Universal Robots PolyScope program: Tall_LidToCamera.urp

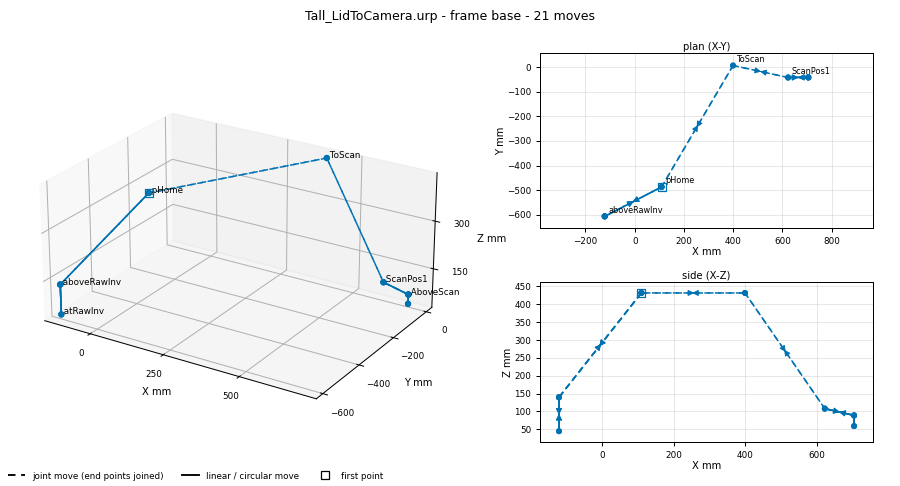
[picture p0: tool path of Tall_LidToCamera.urp in frame base, 21 of 21 moves have a stored position in this frame; points joined in program order, loops and branches not executed]
Program Tall_LidToCamera (installation=admin directory=/programs/THU_530PM/Final createdIn=3.8.0.61336 lastSavedIn=3.15.8.106339 robotSerialNumber=2015350926)
Calibrated DH parameters: a=[0, -0.425, -0.39225, 0, 0, 0]; d=[0.089159, 0, 0, 0.10915, 0.09465, 0.0823]; alpha=[1.570796, 0, 0, 1.570796, -1.570796, 0]; deltaTheta=[0, 0, 0, 0, 0, 0]
Robot Program (runOnlyOnce=true)
  Set DigitalOutput pin=digital_out[0]; digitalValue=0
  MoveJ speed 180 deg/s, acceleration 200 deg/s^2 (useActiveTCP=true)
    Waypoint pHome: TCP in base x=109.083 y=-486.882 z=431.849 mm, rx=0.0001 ry=3.1416 rz=-0.0001 rad; joints [89.992, -90.005, 90.008, -90.008, -90, -0.005] deg
    Call _adminLinearIndex3
    Waypoint aboveRawInv: TCP in base x=-121.783 y=-606.282 z=139.409 mm, rx=2.2212 ry=2.2177 rz=-0.0009 rad; joints [68.458, -61.32, 99.129, -127.902, -89.865, 68.547] deg
  MoveL speed 250 mm/s, acceleration 1200 mm/s^2 (useActiveTCP=true) feature=Base
    Waypoint atRawInv: TCP in base x=-121.765 y=-606.273 z=44.483 mm, rx=2.2211 ry=2.2178 rz=-0.0009 rad; joints [68.459, -52.315, 101.951, -139.731, -89.865, 68.544] deg
    Set DigitalOutput pin=digital_out[0]; digitalValue=1
    Wait Sleep waitTime=1
    Waypoint aboveRawInv: TCP in base x=-121.783 y=-606.282 z=139.409 mm, rx=2.2212 ry=2.2177 rz=-0.0009 rad; joints [68.458, -61.32, 99.129, -127.902, -89.865, 68.547] deg
  MoveJ speed 180 deg/s, acceleration 200 deg/s^2 (useActiveTCP=true)
    Waypoint pHome: TCP in base x=109.083 y=-486.882 z=431.849 mm, rx=0.0001 ry=3.1416 rz=-0.0001 rad; joints [89.992, -90.005, 90.008, -90.008, -90, -0.005] deg
  Call _adminLinearIndex1
  MoveJ speed 60 deg/s, acceleration 80 deg/s^2 (useActiveTCP=true)
    Waypoint ToScan: TCP in base x=399.431 y=6.288 z=431.784 mm, rx=0 ry=-3.1415 rz=0 rad; joints [165.046, -103.944, 102.123, -88.173, -90.001, 75.046] deg
    Waypoint ScanPos1: TCP in base x=623.056 y=-42.326 z=107.794 mm, rx=0.0456 ry=-3.1308 rz=0.0038 rad; joints [166.086, -57.904, 99.074, -130.624, -90.289, 74.42] deg
  MoveL speed 250 mm/s, acceleration 1200 mm/s^2 (useActiveTCP=true) feature=Base
    Waypoint AboveScan: TCP in base x=704.91 y=-41.789 z=88.68 mm, rx=0.0458 ry=-3.1307 rz=0.0039 rad; joints [167.748, -47.56, 83.623, -125.504, -90.275, 76.074] deg
    Waypoint AtScan: TCP in base x=704.921 y=-41.77 z=58.801 mm, rx=0.0456 ry=-3.1306 rz=0.0038 rad; joints [167.749, -45.085, 84.321, -128.675, -90.272, 76.08] deg
    Set DigitalOutput pin=digital_out[0]; digitalValue=0
    Wait Sleep waitTime=1
    Waypoint AboveScan: TCP in base x=704.91 y=-41.789 z=88.68 mm, rx=0.0458 ry=-3.1307 rz=0.0039 rad; joints [167.748, -47.56, 83.623, -125.504, -90.275, 76.074] deg
    Waypoint ScanPos1: TCP in base x=623.056 y=-42.326 z=107.794 mm, rx=0.0456 ry=-3.1308 rz=0.0038 rad; joints [166.086, -57.904, 99.074, -130.624, -90.289, 74.42] deg
    Script file /programs/THU_530PM/vision_pc_modbus.script
      | pc_ip = "10.241.34.37"
      | pc_port = 30002
      | 
      | connection = socket_open(pc_ip, pc_port, "vision_socket")
      | 
      | if (connection):
      |     socket_send_string("run_vision", "vision_socket")
      |     socket_close("vision_socket")
      | end
      | 
      | timeout = 15.0
      | elapsed =0.0
      | visionResult = 0
      | while visionResult == 0 and elapsed < timeout:
      |          sync()
      |          sleep(0.2)
      |          elapsed = elapsed + 0.2
      |          visionResult = modbus_get_signal_status ("vision_result")
      |          sync()
      | end
    Wait Sleep waitTime=2
  MoveJ speed 60 deg/s, acceleration 80 deg/s^2 (useActiveTCP=true)
    Waypoint AboveScan: TCP in base x=704.91 y=-41.789 z=88.68 mm, rx=0.0458 ry=-3.1307 rz=0.0039 rad; joints [167.748, -47.56, 83.623, -125.504, -90.275, 76.074] deg
    Waypoint AtScan: TCP in base x=704.921 y=-41.77 z=58.801 mm, rx=0.0456 ry=-3.1306 rz=0.0038 rad; joints [167.749, -45.085, 84.321, -128.675, -90.272, 76.08] deg
    Set DigitalOutput pin=digital_out[0]; digitalValue=1
    Wait Sleep waitTime=1
    Waypoint AboveScan: TCP in base x=704.91 y=-41.789 z=88.68 mm, rx=0.0458 ry=-3.1307 rz=0.0039 rad; joints [167.748, -47.56, 83.623, -125.504, -90.275, 76.074] deg
  MoveJ speed 60 deg/s, acceleration 80 deg/s^2 (useActiveTCP=true)
    Waypoint ScanPos1: TCP in base x=623.056 y=-42.326 z=107.794 mm, rx=0.0456 ry=-3.1308 rz=0.0038 rad; joints [166.086, -57.904, 99.074, -130.624, -90.289, 74.42] deg
    Waypoint ToScan: TCP in base x=399.431 y=6.288 z=431.784 mm, rx=0 ry=-3.1415 rz=0 rad; joints [165.046, -103.944, 102.123, -88.173, -90.001, 75.046] deg
    Waypoint pHome: TCP in base x=109.083 y=-486.882 z=431.849 mm, rx=0.0001 ry=3.1416 rz=-0.0001 rad; joints [89.992, -90.005, 90.008, -90.008, -90, -0.005] deg
    Call _adminLinearIndex3
    Waypoint aboveRawInv: TCP in base x=-121.783 y=-606.282 z=139.409 mm, rx=2.2212 ry=2.2177 rz=-0.0009 rad; joints [68.458, -61.32, 99.129, -127.902, -89.865, 68.547] deg
  MoveL speed 250 mm/s, acceleration 1200 mm/s^2 (useActiveTCP=true) feature=Base
    Waypoint atRawInv: TCP in base x=-121.765 y=-606.273 z=44.483 mm, rx=2.2211 ry=2.2178 rz=-0.0009 rad; joints [68.459, -52.315, 101.951, -139.731, -89.865, 68.544] deg
    Set DigitalOutput pin=digital_out[0]; digitalValue=0
    Wait Sleep waitTime=1
    Waypoint aboveRawInv: TCP in base x=-121.783 y=-606.282 z=139.409 mm, rx=2.2212 ry=2.2177 rz=-0.0009 rad; joints [68.458, -61.32, 99.129, -127.902, -89.865, 68.547] deg
  MoveJ speed 180 deg/s, acceleration 200 deg/s^2 (useActiveTCP=true)
    Waypoint pHome: TCP in base x=109.083 y=-486.882 z=431.849 mm, rx=0.0001 ry=3.1416 rz=-0.0001 rad; joints [89.992, -90.005, 90.008, -90.008, -90, -0.005] deg
SubProgram -> _adminLinearIndex3
SubProgram  [hidden by the author, left out]
SubProgram _adminLinearIndex3 (keepSynchronizedWithDisk=false) programFile=/programs/me345_admin/_adminLinearIndex3.urp
  Folder Move_linear_slide_Index1
    var_1 := False
    Loop While (checkContinuously=false) expression=var_1≟ False
      var_1 := socket_open("10.241.34.44",4001)
    var_3 := 1
    Send := "s r0x24 21"
    Script: socket_send_string(Send)
    Script: socket_send_byte(13)
    Send_Reply := socket_read_string()
    Send := "s r0xca 103936"
    Script: socket_send_string(Send)
    Script: socket_send_byte(13)
    Send_Reply := socket_read_string()
    Send := "t 1"
    Script: socket_send_string(Send)
    Script: socket_send_byte(13)
    Send_Reply := socket_read_string()
    Loop While (checkContinuously=false) expression=var_3≠0
      Send := "g r0xA0"
      Script: socket_send_string(Send)
      Script: socket_send_byte(13)
      var_3 := socket_get_var("v")
      Wait Sleep waitTime=0.1
    Script: socket_close()
    Script: sync()
SubProgram _adminLinearIndex1 [hidden by the author, left out]
